TYPE ST_Widget_Plug_Template :
STRUCT
	sDisplayName	: STRING := ''; // Insert STRING here to overwrite iot.DisplayName

	bOn				: BOOL;

	sMode			: STRING; // can be set to any value, does not have to match the array below
	aModes			: ARRAY[0..1] OF STRING;
END_STRUCT
END_TYPE

(* stored: Version 1.1.0.1, ProductVersion 3.1.4024.11
   DUT ST_Widget_Plug_Template: Id {8a9a2dc5-384f-4f1a-9376-b2f014433b52} *)
